// TIA Portal V17 export
// export: Created 2025-03-07T09:18:53.7752004Z, ExportSetting WithDefaults, DisplayName Totally Integrated Automation Portal, DisplayVersion V17 Update 8, DisplayName TIA Portal Openness, DisplayVersion V17 Update 8, DisplayName TIA Portal Version Control Interface, DisplayVersion V17, DisplayName SINAMICS Startdrive Advanced, DisplayVersion V17 SP2, DisplayName SINAMICS Startdrive G110M, G120, G120C, G120D, G120P, G115D, DisplayVersion V17 SP2, DisplayName SINAMICS Startdrive G130, G150, S120, S150, SINAMICS MV, S210, DisplayVersion V17 SP2, DisplayName STEP 7 Professional, DisplayVersion V17 Update 8, DisplayName SINUMERIK ONE STEP 7 Toolbox, DisplayVersion V17 Update 12, DisplayName SINUMERIK 840D sl STEP 7 Toolbox, DisplayVersion V17 Update 12, DisplayName STEP 7 Safety, DisplayVersion V17 Update 6, DisplayName WinCC Advanced, DisplayVersion V17 Update 8
FUNCTION_BLOCK "FB20200_TRUMPF_READY"   // FB20200, LAD
TITLE = FB20200 READY TRUMPF
{ S7_Optimized_Access := 'FALSE' }
VERSION : 0.1
// stored: AutoNumber false, IsIECCheckEnabled false, SetENOAutomatically false, UDAEnableTagReadback false
   VAR_INPUT
      iLIMIT_MIN_POWER : Int;   // LASER POWER MIN LIMIT
      iLIMIT_MAX_POWER : Int;   // LASER POWER MAX LIMIT
      iCOMMAND_POWER : Int;   // CNC POWER VALUE
      iCOMMAND_PROCESSING : Int;   // CNC PROCESSING VALUE
      iCOMMAND_POWER_PORTION_CORE : Int;   // CNC POWER PORTION CORE VALUE
      iSTATUS_READY_LASER_READY : Bool;   // LASER STATUS: READY
      iLASER_IS_ON : Bool;   // LASER IS ON
      iSYSTEM_ERROR_LASER_FAULT : Bool;   // LASER SYSTEM ERROR / FAULT
      iEXTERNAL_CONTROL_READY : Bool;   // LASER EXTERNAL CONTROL READY
      iPROGRAM_ACTIVE : Bool;   // LASER PROGRAM ACTIVE
      iSOURCE_ENABLED : Bool;   // -
      iCOOLING_UNIT_FLOW_PRESENT : Bool;
      iCOOLING_UNIT_OVERTEMPERATURE : Bool;
      iLASER_ENABLE_POWER_SEQ : Bool;   // -
      iLASER_DISABLE_POWER_SEQ : Bool;   // -
      iSAFETY_GATES_CLOSED_LOCKED : Bool;   // LOCAL SAFETY GATES CLOSED AND LOCKED
      iLASER_ASSIGNED : Bool;   // LASER ASSIGNED
      iMACHINE_ON : Bool;   // LOCAL MACHINE ON
      iMACHINE_ON_DELAYED : Bool;   // LOCAL MACHINE ON DELAYED
      iLASER_READY_F_CIRCUIT_BRAKER : Bool;   // LASER CIRCUIT BREAKER OK
      iLASER_WARNING_LAP_ON : Bool;   // LOCAL STATION UNIT ANY CYCLE ACTIVE
      iSTATION_UNIT_ANY_CYCLE_ACT : Bool;   // LASER ACTIVE DB START GENERAL CONDITIONS
      iLASER_ACT_START_GEN_CONDITION : Bool;
      iUNIT_NO : Byte;
   END_VAR
   VAR_OUTPUT
      oLIGHT_PATH : Byte;
      oPROGRAM_NUMBER : Byte;
      oPOWER_VALUE : DInt;
      oPROCESSING_VALUE : DInt;
      oPOWER_PORTION_CORE_VALUE : DInt;
      oLASER_RESET_FAULT_ERROR : Bool;
      oLASER_REQUEST : Bool;
      oEXTERNAL_CONTROL : Bool;
      oLASER_ON : Bool;
      oLASER_ARM : Bool;
      oSTATION_RHP_SEOC_ALARMS : Bool;
      oSTATION_WARNING : Bool;
      oREADY_TO_EMISSION : Bool;
      oALARM_CIRCUIT_BREAKER_ALARM : Bool;
      oALARM_LASER_ERROR : Bool;
      oALARM_WARNING_LASER : Bool;
      oALARM_LASER_NOT_READY : Bool;
      oALARM_LASER_NOT_SWITCHED_ON : Bool;
      oALARM_ANALOG_CONTROL_ERROR : Bool;
      oALARM_LASER_NOT_ASSIGNED : Bool;
      oALARM_OVERTEMPERATURE_ALARM : Bool;
      oALARM_LASER_EMERGENCY_STOP_ACTIVE : Bool;
      oALARM_LASER_SC_STATUS_ACTIVE : Bool;
      oALARM_ACTIVE_PANEL_ERROR : Bool;
      oALARM_LASER_MODULE_1_IN_TEST_MODE : Bool;
      oALARM_FAULT : Bool;
   END_VAR
   VAR DB_SPECIFIC
      DATA { S7_SetPoint := 'True'} : "LASER READY";
      "EXT PULSE START REQ" { S7_SetPoint := 'True'} : TON_TIME;
      "COOLING UNIT FLOW IN" : Bool;
      "COOLING OVERTEMPERATURE IN" : Bool;
      "COOLING UNIT FLOW ALARM" : Bool;
      "COOLING OVERTEMPERATURE ALARM" : Bool;
      INT_AUX : Int;
   END_VAR
   VAR_TEMP
      DB_NUMBER : DInt;
   END_VAR
   VAR_TEMP   // added for the SCL form of the ladder/FBD networks
      _w1 : Bool;
      _w2 : Bool;
      _w3 : Bool;
      _w4 : Bool;
   END_VAR
BEGIN

NETWORK
TITLE = READ INSTANCE DB NUMBER
      L     DINO;
      +     10#800000;
      T     #DB_NUMBER;

REGION Network 2: VARIABLE VALUE
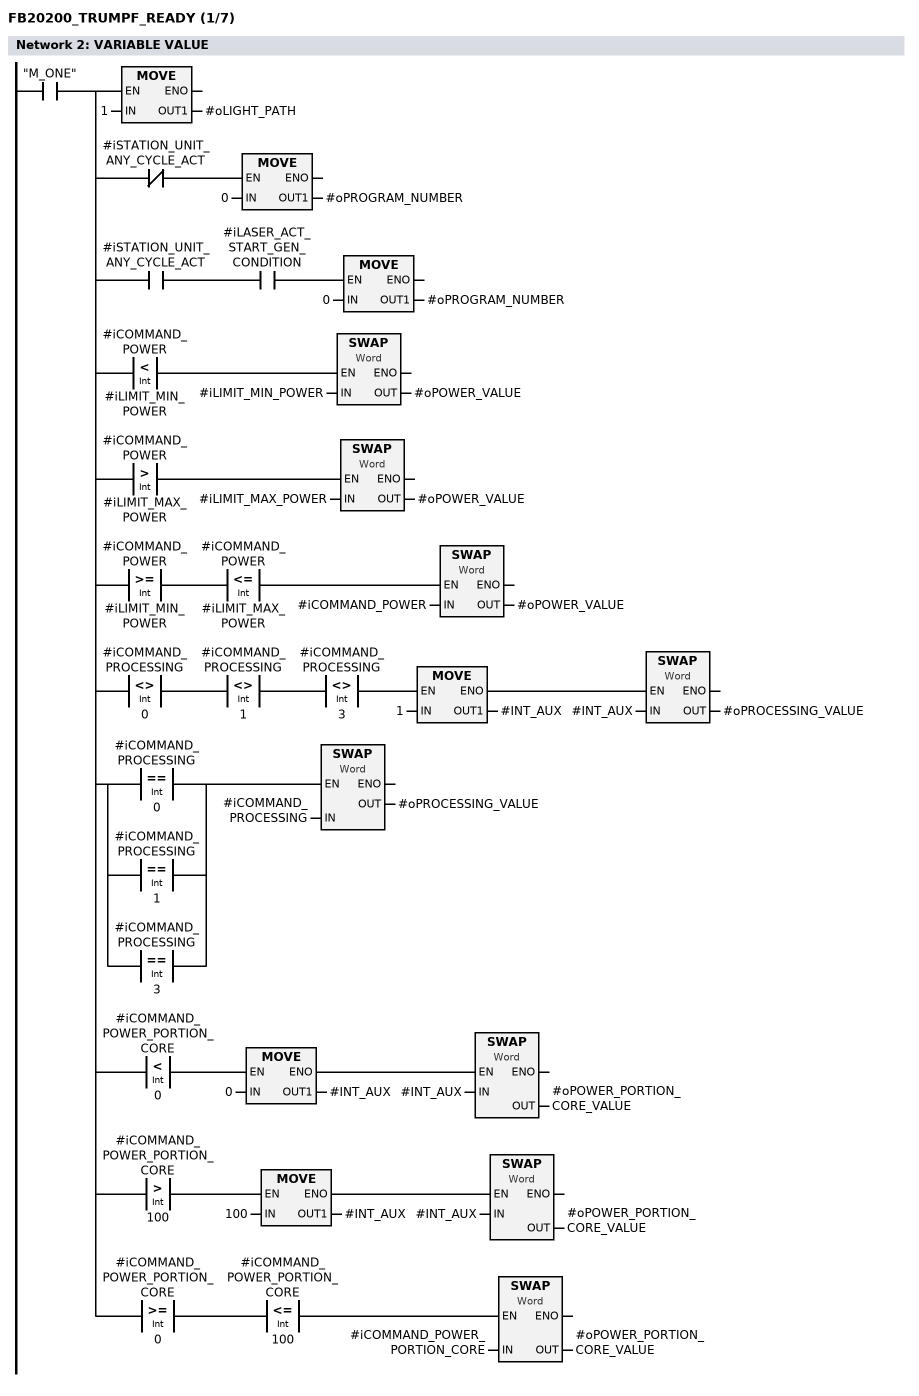
   IF "M_ONE" THEN #oLIGHT_PATH := 1; END_IF;
   IF "M_ONE" AND NOT #iSTATION_UNIT_ANY_CYCLE_ACT THEN #oPROGRAM_NUMBER := 0; END_IF;
   IF "M_ONE" AND #iSTATION_UNIT_ANY_CYCLE_ACT AND #iLASER_ACT_START_GEN_CONDITION THEN
       #oPROGRAM_NUMBER := 0;
   END_IF;
   IF "M_ONE" AND (#iCOMMAND_POWER < #iLIMIT_MIN_POWER) THEN
       #oPOWER_VALUE := SWAP(#iLIMIT_MIN_POWER);
   END_IF;
   IF "M_ONE" AND (#iCOMMAND_POWER > #iLIMIT_MAX_POWER) THEN
       #oPOWER_VALUE := SWAP(#iLIMIT_MAX_POWER);
   END_IF;
   IF "M_ONE" AND (#iCOMMAND_POWER >= #iLIMIT_MIN_POWER) AND (#iCOMMAND_POWER <= #iLIMIT_MAX_POWER) THEN
       #oPOWER_VALUE := SWAP(#iCOMMAND_POWER);
   END_IF;
   IF "M_ONE" AND (#iCOMMAND_PROCESSING <> 0) AND (#iCOMMAND_PROCESSING <> 1) AND (#iCOMMAND_PROCESSING <> 3) THEN
       #INT_AUX := 1;
       #oPROCESSING_VALUE := SWAP(#INT_AUX);
   END_IF;
   IF "M_ONE" AND ((#iCOMMAND_PROCESSING = 0) OR (#iCOMMAND_PROCESSING = 1) OR (#iCOMMAND_PROCESSING = 3)) THEN
       #oPROCESSING_VALUE := SWAP(#iCOMMAND_PROCESSING);
   END_IF;
   IF "M_ONE" AND (#iCOMMAND_POWER_PORTION_CORE < 0) THEN
       #INT_AUX := 0;
       #oPOWER_PORTION_CORE_VALUE := SWAP(#INT_AUX);
   END_IF;
   IF "M_ONE" AND (#iCOMMAND_POWER_PORTION_CORE > 100) THEN
       #INT_AUX := 100;
       #oPOWER_PORTION_CORE_VALUE := SWAP(#INT_AUX);
   END_IF;
   IF "M_ONE" AND (#iCOMMAND_POWER_PORTION_CORE >= 0) AND (#iCOMMAND_POWER_PORTION_CORE <= 100) THEN
       #oPOWER_PORTION_CORE_VALUE := SWAP(#iCOMMAND_POWER_PORTION_CORE);
   END_IF;
END_REGION

REGION Network 3: INPUT
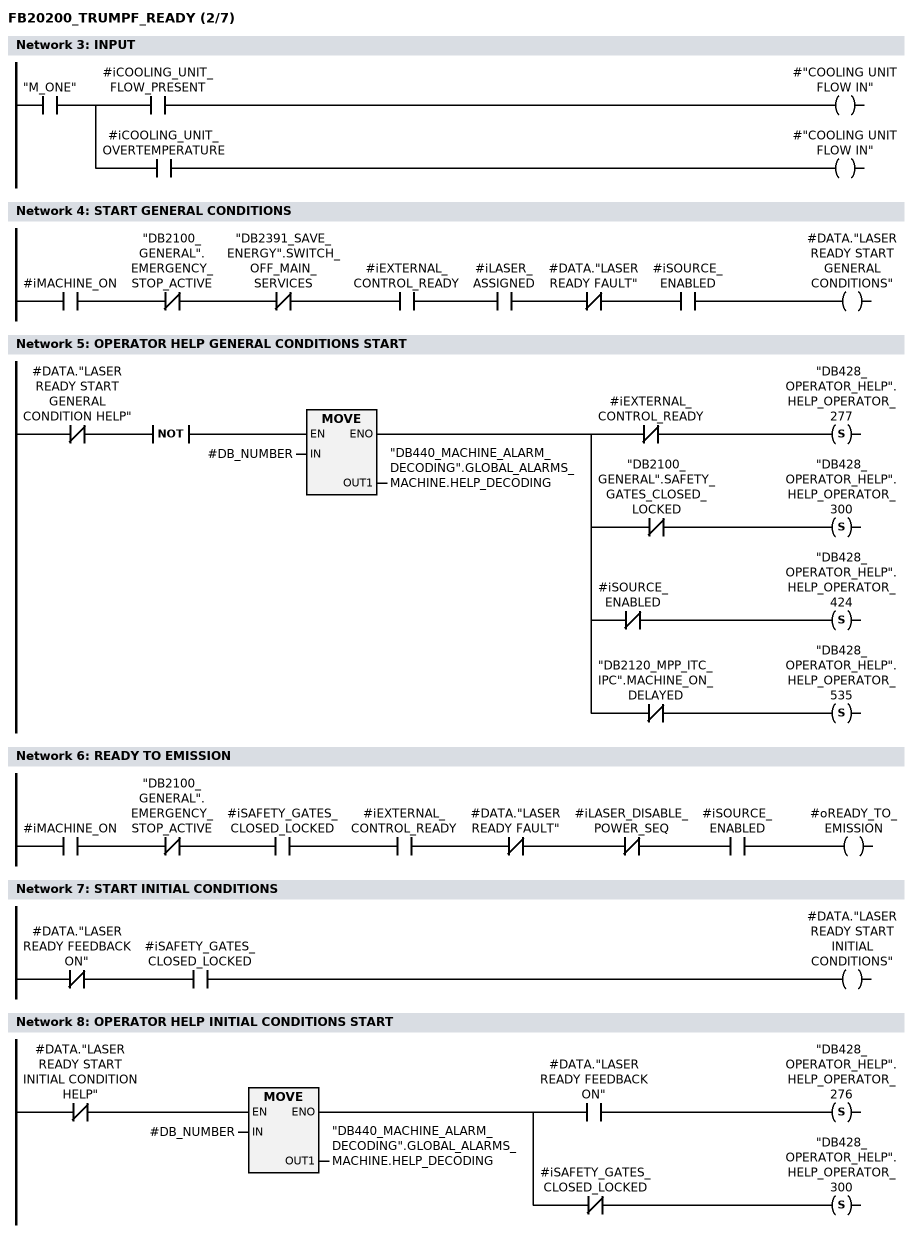
   RUNG wire#powerrail
      Contact( "M_ONE" )
      wire#w1
      Contact( #iCOOLING_UNIT_FLOW_PRESENT )
      Coil( #"COOLING UNIT FLOW IN" )
   END_RUNG
   RUNG wire#w1
      Contact( #iCOOLING_UNIT_OVERTEMPERATURE )
      Coil( #"COOLING UNIT FLOW IN" )
   END_RUNG
   // the same network as SCL:
   #"COOLING UNIT FLOW IN" := "M_ONE" AND #iCOOLING_UNIT_FLOW_PRESENT;
   #"COOLING UNIT FLOW IN" := "M_ONE" AND #iCOOLING_UNIT_OVERTEMPERATURE;
END_REGION

REGION Network 4: START GENERAL CONDITIONS
   RUNG wire#powerrail
      Contact( #iMACHINE_ON )
      I_Contact( "DB2100_GENERAL".EMERGENCY_STOP_ACTIVE )
      I_Contact( "DB2391_SAVE_ENERGY".SWITCH_OFF_MAIN_SERVICES )
      Contact( #iEXTERNAL_CONTROL_READY )
      Contact( #iLASER_ASSIGNED )
      I_Contact( #DATA."LASER READY FAULT" )
      Contact( #iSOURCE_ENABLED )
      Coil( #DATA."LASER READY START GENERAL CONDITIONS" )
   END_RUNG
   // the same network as SCL:
   #DATA."LASER READY START GENERAL CONDITIONS" := #iMACHINE_ON AND NOT "DB2100_GENERAL".EMERGENCY_STOP_ACTIVE AND NOT "DB2391_SAVE_ENERGY".SWITCH_OFF_MAIN_SERVICES AND #iEXTERNAL_CONTROL_READY AND #iLASER_ASSIGNED AND NOT #DATA."LASER READY FAULT" AND #iSOURCE_ENABLED;
END_REGION

REGION Network 5: OPERATOR HELP GENERAL CONDITIONS START
   RUNG wire#powerrail
      I_Contact( #DATA."LASER READY START GENERAL CONDITION HELP" )
      Not()
      Move(in := #DB_NUMBER, out1 => "DB440_MACHINE_ALARM_DECODING".GLOBAL_ALARMS_MACHINE.HELP_DECODING)
      wire#w1
      I_Contact( #iEXTERNAL_CONTROL_READY )
      S_Coil( "DB428_OPERATOR_HELP".HELP_OPERATOR_277 )
   END_RUNG
   RUNG wire#w1
      I_Contact( "DB2100_GENERAL".SAFETY_GATES_CLOSED_LOCKED )
      S_Coil( "DB428_OPERATOR_HELP".HELP_OPERATOR_300 )
   END_RUNG
   RUNG wire#w1
      I_Contact( #iSOURCE_ENABLED )
      S_Coil( "DB428_OPERATOR_HELP".HELP_OPERATOR_424 )
   END_RUNG
   RUNG wire#w1
      I_Contact( "DB2120_MPP_ITC_IPC".MACHINE_ON_DELAYED )
      S_Coil( "DB428_OPERATOR_HELP".HELP_OPERATOR_535 )
   END_RUNG
   // the same network as SCL:
   #_w1 := NOT (NOT #DATA."LASER READY START GENERAL CONDITION HELP");
   IF #_w1 THEN "DB440_MACHINE_ALARM_DECODING".GLOBAL_ALARMS_MACHINE.HELP_DECODING := #DB_NUMBER; END_IF;
   IF #_w1 AND NOT #iEXTERNAL_CONTROL_READY THEN "DB428_OPERATOR_HELP".HELP_OPERATOR_277 := TRUE; END_IF;
   IF #_w1 AND NOT "DB2100_GENERAL".SAFETY_GATES_CLOSED_LOCKED THEN
       "DB428_OPERATOR_HELP".HELP_OPERATOR_300 := TRUE;
   END_IF;
   IF #_w1 AND NOT #iSOURCE_ENABLED THEN "DB428_OPERATOR_HELP".HELP_OPERATOR_424 := TRUE; END_IF;
   IF #_w1 AND NOT "DB2120_MPP_ITC_IPC".MACHINE_ON_DELAYED THEN
       "DB428_OPERATOR_HELP".HELP_OPERATOR_535 := TRUE;
   END_IF;
END_REGION

REGION Network 6: READY TO EMISSION
   RUNG wire#powerrail
      Contact( #iMACHINE_ON )
      I_Contact( "DB2100_GENERAL".EMERGENCY_STOP_ACTIVE )
      Contact( #iSAFETY_GATES_CLOSED_LOCKED )
      Contact( #iEXTERNAL_CONTROL_READY )
      I_Contact( #DATA."LASER READY FAULT" )
      I_Contact( #iLASER_DISABLE_POWER_SEQ )
      Contact( #iSOURCE_ENABLED )
      Coil( #oREADY_TO_EMISSION )
   END_RUNG
   // the same network as SCL:
   #oREADY_TO_EMISSION := #iMACHINE_ON AND NOT "DB2100_GENERAL".EMERGENCY_STOP_ACTIVE AND #iSAFETY_GATES_CLOSED_LOCKED AND #iEXTERNAL_CONTROL_READY AND NOT #DATA."LASER READY FAULT" AND NOT #iLASER_DISABLE_POWER_SEQ AND #iSOURCE_ENABLED;
END_REGION

REGION Network 7: START INITIAL CONDITIONS
   RUNG wire#powerrail
      I_Contact( #DATA."LASER READY FEEDBACK ON" )
      Contact( #iSAFETY_GATES_CLOSED_LOCKED )
      Coil( #DATA."LASER READY START INITIAL CONDITIONS" )
   END_RUNG
   // the same network as SCL:
   #DATA."LASER READY START INITIAL CONDITIONS" := NOT #DATA."LASER READY FEEDBACK ON" AND #iSAFETY_GATES_CLOSED_LOCKED;
END_REGION

REGION Network 8: OPERATOR HELP INITIAL CONDITIONS START
   RUNG wire#powerrail
      I_Contact( #DATA."LASER READY START INITIAL CONDITION HELP" )
      Move(in := #DB_NUMBER, out1 => "DB440_MACHINE_ALARM_DECODING".GLOBAL_ALARMS_MACHINE.HELP_DECODING)
      wire#w1
      Contact( #DATA."LASER READY FEEDBACK ON" )
      S_Coil( "DB428_OPERATOR_HELP".HELP_OPERATOR_276 )
   END_RUNG
   RUNG wire#w1
      I_Contact( #iSAFETY_GATES_CLOSED_LOCKED )
      S_Coil( "DB428_OPERATOR_HELP".HELP_OPERATOR_300 )
   END_RUNG
   // the same network as SCL:
   #_w1 := NOT #DATA."LASER READY START INITIAL CONDITION HELP";
   IF #_w1 THEN "DB440_MACHINE_ALARM_DECODING".GLOBAL_ALARMS_MACHINE.HELP_DECODING := #DB_NUMBER; END_IF;
   IF #_w1 AND #DATA."LASER READY FEEDBACK ON" THEN "DB428_OPERATOR_HELP".HELP_OPERATOR_276 := TRUE; END_IF;
   IF #_w1 AND NOT #iSAFETY_GATES_CLOSED_LOCKED THEN "DB428_OPERATOR_HELP".HELP_OPERATOR_300 := TRUE; END_IF;
END_REGION

REGION Network 9: AUTO START REQUEST
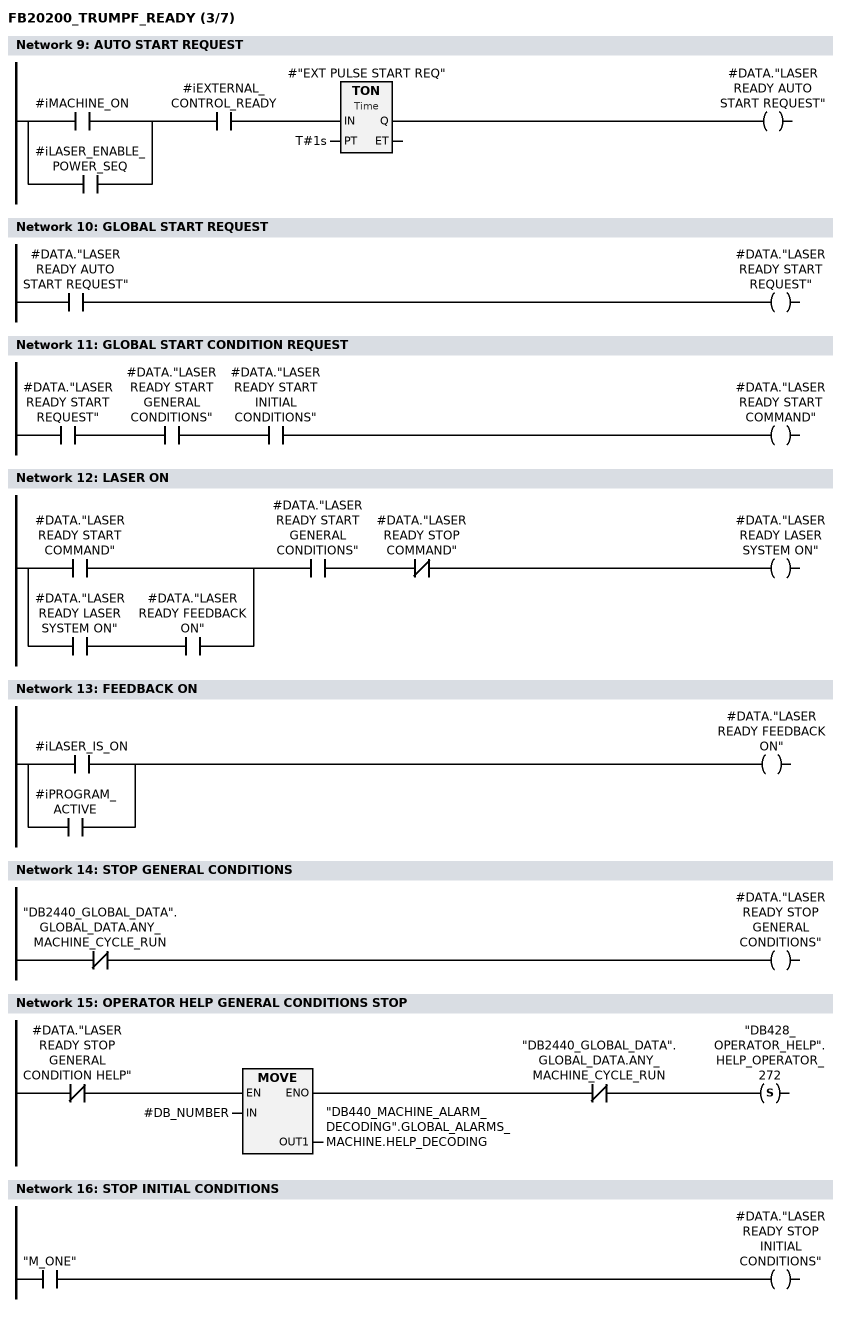
   RUNG wire#powerrail
      Contact( #iMACHINE_ON )
      wire#w1
      Contact( #iEXTERNAL_CONTROL_READY )
      { S7_Templates := "time_type := Time" } #"EXT PULSE START REQ".TON(pt := T#1s, et =>)
      Coil( #DATA."LASER READY AUTO START REQUEST" )
   END_RUNG
   RUNG wire#powerrail
      Contact( #iLASER_ENABLE_POWER_SEQ )
   END_RUNG wire#w1
   // the same network as SCL:
   #"EXT PULSE START REQ"(IN := (#iMACHINE_ON OR #iLASER_ENABLE_POWER_SEQ) AND #iEXTERNAL_CONTROL_READY,   // TON
                          PT := T#1s);
   #DATA."LASER READY AUTO START REQUEST" := #"EXT PULSE START REQ".Q;
END_REGION

REGION Network 10: GLOBAL START REQUEST
   RUNG wire#powerrail
      Contact( #DATA."LASER READY AUTO START REQUEST" )
      Coil( #DATA."LASER READY START REQUEST" )
   END_RUNG
   // the same network as SCL:
   #DATA."LASER READY START REQUEST" := #DATA."LASER READY AUTO START REQUEST";
END_REGION

REGION Network 11: GLOBAL START CONDITION REQUEST
   RUNG wire#powerrail
      Contact( #DATA."LASER READY START REQUEST" )
      Contact( #DATA."LASER READY START GENERAL CONDITIONS" )
      Contact( #DATA."LASER READY START INITIAL CONDITIONS" )
      Coil( #DATA."LASER READY START COMMAND" )
   END_RUNG
   // the same network as SCL:
   #DATA."LASER READY START COMMAND" := #DATA."LASER READY START REQUEST" AND #DATA."LASER READY START GENERAL CONDITIONS" AND #DATA."LASER READY START INITIAL CONDITIONS";
END_REGION

REGION Network 12: LASER ON
   RUNG wire#powerrail
      Contact( #DATA."LASER READY START COMMAND" )
      wire#w1
      Contact( #DATA."LASER READY START GENERAL CONDITIONS" )
      I_Contact( #DATA."LASER READY STOP COMMAND" )
      Coil( #DATA."LASER READY LASER SYSTEM ON" )
   END_RUNG
   RUNG wire#powerrail
      Contact( #DATA."LASER READY LASER SYSTEM ON" )
      Contact( #DATA."LASER READY FEEDBACK ON" )
   END_RUNG wire#w1
   // the same network as SCL:
   #DATA."LASER READY LASER SYSTEM ON" := (#DATA."LASER READY START COMMAND" OR (#DATA."LASER READY LASER SYSTEM ON" AND #DATA."LASER READY FEEDBACK ON")) AND #DATA."LASER READY START GENERAL CONDITIONS" AND NOT #DATA."LASER READY STOP COMMAND";
END_REGION

REGION Network 13: FEEDBACK ON
   RUNG wire#powerrail
      Contact( #iLASER_IS_ON )
      wire#w1
      Coil( #DATA."LASER READY FEEDBACK ON" )
   END_RUNG
   RUNG wire#powerrail
      Contact( #iPROGRAM_ACTIVE )
   END_RUNG wire#w1
   // the same network as SCL:
   #DATA."LASER READY FEEDBACK ON" := #iLASER_IS_ON OR #iPROGRAM_ACTIVE;
END_REGION

REGION Network 14: STOP GENERAL CONDITIONS
   RUNG wire#powerrail
      I_Contact( "DB2440_GLOBAL_DATA".GLOBAL_DATA.ANY_MACHINE_CYCLE_RUN )
      Coil( #DATA."LASER READY STOP GENERAL CONDITIONS" )
   END_RUNG
   // the same network as SCL:
   #DATA."LASER READY STOP GENERAL CONDITIONS" := NOT "DB2440_GLOBAL_DATA".GLOBAL_DATA.ANY_MACHINE_CYCLE_RUN;
END_REGION

REGION Network 15: OPERATOR HELP GENERAL CONDITIONS STOP
   RUNG wire#powerrail
      I_Contact( #DATA."LASER READY STOP GENERAL CONDITION HELP" )
      Move(in := #DB_NUMBER, out1 => "DB440_MACHINE_ALARM_DECODING".GLOBAL_ALARMS_MACHINE.HELP_DECODING)
      I_Contact( "DB2440_GLOBAL_DATA".GLOBAL_DATA.ANY_MACHINE_CYCLE_RUN )
      S_Coil( "DB428_OPERATOR_HELP".HELP_OPERATOR_272 )
   END_RUNG
   // the same network as SCL:
   #_w1 := NOT #DATA."LASER READY STOP GENERAL CONDITION HELP";
   IF #_w1 THEN "DB440_MACHINE_ALARM_DECODING".GLOBAL_ALARMS_MACHINE.HELP_DECODING := #DB_NUMBER; END_IF;
   IF #_w1 AND NOT "DB2440_GLOBAL_DATA".GLOBAL_DATA.ANY_MACHINE_CYCLE_RUN THEN
       "DB428_OPERATOR_HELP".HELP_OPERATOR_272 := TRUE;
   END_IF;
END_REGION

REGION Network 16: STOP INITIAL CONDITIONS
   RUNG wire#powerrail
      Contact( "M_ONE" )
      Coil( #DATA."LASER READY STOP INITIAL CONDITIONS" )
   END_RUNG
   // the same network as SCL:
   #DATA."LASER READY STOP INITIAL CONDITIONS" := "M_ONE";
END_REGION

REGION Network 17: OPERATOR HELP INITIAL CONDITIONS STOP
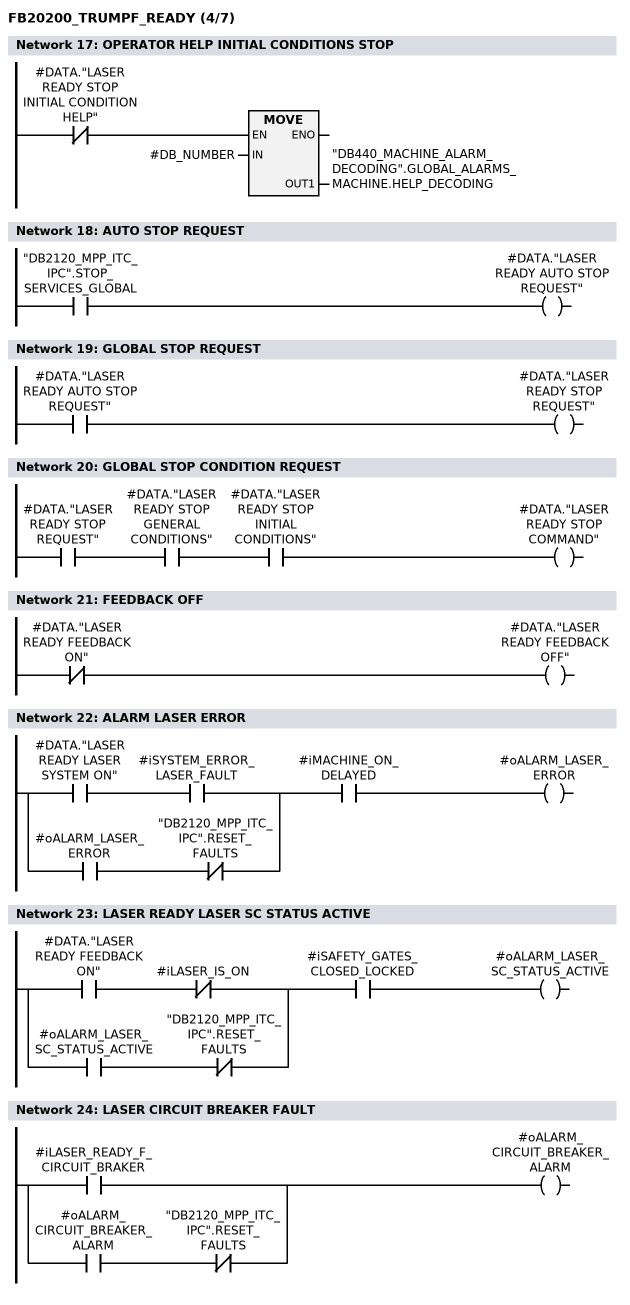
   RUNG wire#powerrail
      I_Contact( #DATA."LASER READY STOP INITIAL CONDITION HELP" )
      Move(in := #DB_NUMBER, out1 => "DB440_MACHINE_ALARM_DECODING".GLOBAL_ALARMS_MACHINE.HELP_DECODING)
   END_RUNG
   // the same network as SCL:
   IF NOT #DATA."LASER READY STOP INITIAL CONDITION HELP" THEN
       "DB440_MACHINE_ALARM_DECODING".GLOBAL_ALARMS_MACHINE.HELP_DECODING := #DB_NUMBER;
   END_IF;
END_REGION

REGION Network 18: AUTO STOP REQUEST
   RUNG wire#powerrail
      Contact( "DB2120_MPP_ITC_IPC".STOP_SERVICES_GLOBAL )
      Coil( #DATA."LASER READY AUTO STOP REQUEST" )
   END_RUNG
   // the same network as SCL:
   #DATA."LASER READY AUTO STOP REQUEST" := "DB2120_MPP_ITC_IPC".STOP_SERVICES_GLOBAL;
END_REGION

REGION Network 19: GLOBAL STOP REQUEST
   RUNG wire#powerrail
      Contact( #DATA."LASER READY AUTO STOP REQUEST" )
      Coil( #DATA."LASER READY STOP REQUEST" )
   END_RUNG
   // the same network as SCL:
   #DATA."LASER READY STOP REQUEST" := #DATA."LASER READY AUTO STOP REQUEST";
END_REGION

REGION Network 20: GLOBAL STOP CONDITION REQUEST
   RUNG wire#powerrail
      Contact( #DATA."LASER READY STOP REQUEST" )
      Contact( #DATA."LASER READY STOP GENERAL CONDITIONS" )
      Contact( #DATA."LASER READY STOP INITIAL CONDITIONS" )
      Coil( #DATA."LASER READY STOP COMMAND" )
   END_RUNG
   // the same network as SCL:
   #DATA."LASER READY STOP COMMAND" := #DATA."LASER READY STOP REQUEST" AND #DATA."LASER READY STOP GENERAL CONDITIONS" AND #DATA."LASER READY STOP INITIAL CONDITIONS";
END_REGION

REGION Network 21: FEEDBACK OFF
   RUNG wire#powerrail
      I_Contact( #DATA."LASER READY FEEDBACK ON" )
      Coil( #DATA."LASER READY FEEDBACK OFF" )
   END_RUNG
   // the same network as SCL:
   #DATA."LASER READY FEEDBACK OFF" := NOT #DATA."LASER READY FEEDBACK ON";
END_REGION

REGION Network 22: ALARM LASER ERROR
   RUNG wire#powerrail
      Contact( #DATA."LASER READY LASER SYSTEM ON" )
      Contact( #iSYSTEM_ERROR_LASER_FAULT )
      wire#w1
      Contact( #iMACHINE_ON_DELAYED )
      Coil( #oALARM_LASER_ERROR )
   END_RUNG
   RUNG wire#powerrail
      Contact( #oALARM_LASER_ERROR )
      I_Contact( "DB2120_MPP_ITC_IPC".RESET_FAULTS )
   END_RUNG wire#w1
   // the same network as SCL:
   #oALARM_LASER_ERROR := ((#DATA."LASER READY LASER SYSTEM ON" AND #iSYSTEM_ERROR_LASER_FAULT) OR (#oALARM_LASER_ERROR AND NOT "DB2120_MPP_ITC_IPC".RESET_FAULTS)) AND #iMACHINE_ON_DELAYED;
END_REGION

REGION Network 23: LASER READY LASER SC STATUS ACTIVE
   RUNG wire#powerrail
      Contact( #DATA."LASER READY FEEDBACK ON" )
      I_Contact( #iLASER_IS_ON )
      wire#w1
      Contact( #iSAFETY_GATES_CLOSED_LOCKED )
      Coil( #oALARM_LASER_SC_STATUS_ACTIVE )
   END_RUNG
   RUNG wire#powerrail
      Contact( #oALARM_LASER_SC_STATUS_ACTIVE )
      I_Contact( "DB2120_MPP_ITC_IPC".RESET_FAULTS )
   END_RUNG wire#w1
   // the same network as SCL:
   #oALARM_LASER_SC_STATUS_ACTIVE := ((#DATA."LASER READY FEEDBACK ON" AND NOT #iLASER_IS_ON) OR (#oALARM_LASER_SC_STATUS_ACTIVE AND NOT "DB2120_MPP_ITC_IPC".RESET_FAULTS)) AND #iSAFETY_GATES_CLOSED_LOCKED;
END_REGION

REGION Network 24: LASER CIRCUIT BREAKER FAULT
   RUNG wire#powerrail
      Contact( #iLASER_READY_F_CIRCUIT_BRAKER )
      wire#w1
      Coil( #oALARM_CIRCUIT_BREAKER_ALARM )
   END_RUNG
   RUNG wire#powerrail
      Contact( #oALARM_CIRCUIT_BREAKER_ALARM )
      I_Contact( "DB2120_MPP_ITC_IPC".RESET_FAULTS )
   END_RUNG wire#w1
   // the same network as SCL:
   #oALARM_CIRCUIT_BREAKER_ALARM := #iLASER_READY_F_CIRCUIT_BRAKER OR (#oALARM_CIRCUIT_BREAKER_ALARM AND NOT "DB2120_MPP_ITC_IPC".RESET_FAULTS);
END_REGION

REGION Network 25: LASER NOT READY
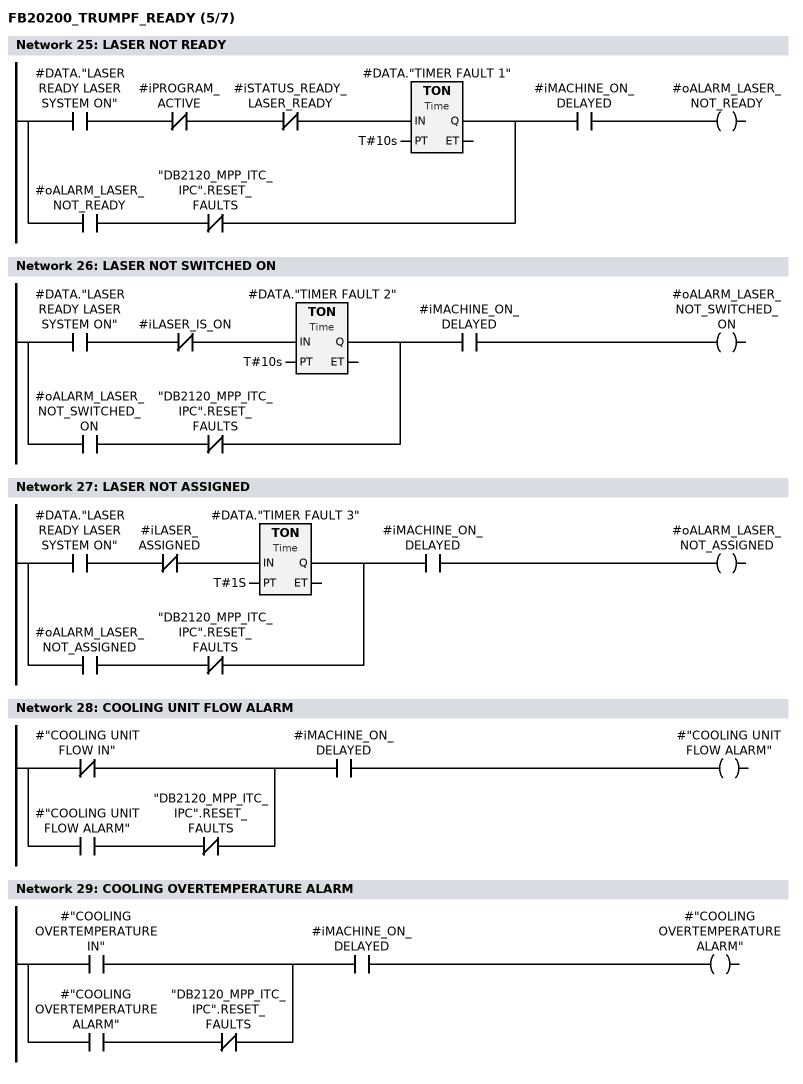
   RUNG wire#powerrail
      Contact( #DATA."LASER READY LASER SYSTEM ON" )
      I_Contact( #iPROGRAM_ACTIVE )
      I_Contact( #iSTATUS_READY_LASER_READY )
      { S7_Templates := "time_type := Time" } #DATA."TIMER FAULT 1".TON(pt := T#10s, et =>)
      wire#w1
      Contact( #iMACHINE_ON_DELAYED )
      Coil( #oALARM_LASER_NOT_READY )
   END_RUNG
   RUNG wire#powerrail
      Contact( #oALARM_LASER_NOT_READY )
      I_Contact( "DB2120_MPP_ITC_IPC".RESET_FAULTS )
   END_RUNG wire#w1
   // the same network as SCL:
   #DATA."TIMER FAULT 1".TON(IN := #DATA."LASER READY LASER SYSTEM ON" AND NOT #iPROGRAM_ACTIVE AND NOT #iSTATUS_READY_LASER_READY,
                           PT := T#10s);
   #oALARM_LASER_NOT_READY := (#DATA."TIMER FAULT 1".Q OR (#oALARM_LASER_NOT_READY AND NOT "DB2120_MPP_ITC_IPC".RESET_FAULTS)) AND #iMACHINE_ON_DELAYED;
END_REGION

REGION Network 26: LASER NOT SWITCHED ON
   RUNG wire#powerrail
      Contact( #DATA."LASER READY LASER SYSTEM ON" )
      I_Contact( #iLASER_IS_ON )
      { S7_Templates := "time_type := Time" } #DATA."TIMER FAULT 2".TON(pt := T#10s, et =>)
      wire#w1
      Contact( #iMACHINE_ON_DELAYED )
      Coil( #oALARM_LASER_NOT_SWITCHED_ON )
   END_RUNG
   RUNG wire#powerrail
      Contact( #oALARM_LASER_NOT_SWITCHED_ON )
      I_Contact( "DB2120_MPP_ITC_IPC".RESET_FAULTS )
   END_RUNG wire#w1
   // the same network as SCL:
   #DATA."TIMER FAULT 2".TON(IN := #DATA."LASER READY LASER SYSTEM ON" AND NOT #iLASER_IS_ON, PT := T#10s);
   #oALARM_LASER_NOT_SWITCHED_ON := (#DATA."TIMER FAULT 2".Q OR (#oALARM_LASER_NOT_SWITCHED_ON AND NOT "DB2120_MPP_ITC_IPC".RESET_FAULTS)) AND #iMACHINE_ON_DELAYED;
END_REGION

REGION Network 27: LASER NOT ASSIGNED
   RUNG wire#powerrail
      Contact( #DATA."LASER READY LASER SYSTEM ON" )
      I_Contact( #iLASER_ASSIGNED )
      { S7_Templates := "time_type := Time" } #DATA."TIMER FAULT 3".TON(pt := T#1S, et =>)
      wire#w1
      Contact( #iMACHINE_ON_DELAYED )
      Coil( #oALARM_LASER_NOT_ASSIGNED )
   END_RUNG
   RUNG wire#powerrail
      Contact( #oALARM_LASER_NOT_ASSIGNED )
      I_Contact( "DB2120_MPP_ITC_IPC".RESET_FAULTS )
   END_RUNG wire#w1
   // the same network as SCL:
   #DATA."TIMER FAULT 3".TON(IN := #DATA."LASER READY LASER SYSTEM ON" AND NOT #iLASER_ASSIGNED, PT := T#1S);
   #oALARM_LASER_NOT_ASSIGNED := (#DATA."TIMER FAULT 3".Q OR (#oALARM_LASER_NOT_ASSIGNED AND NOT "DB2120_MPP_ITC_IPC".RESET_FAULTS)) AND #iMACHINE_ON_DELAYED;
END_REGION

REGION Network 28: COOLING UNIT FLOW ALARM
   RUNG wire#powerrail
      I_Contact( #"COOLING UNIT FLOW IN" )
      wire#w1
      Contact( #iMACHINE_ON_DELAYED )
      Coil( #"COOLING UNIT FLOW ALARM" )
   END_RUNG
   RUNG wire#powerrail
      Contact( #"COOLING UNIT FLOW ALARM" )
      I_Contact( "DB2120_MPP_ITC_IPC".RESET_FAULTS )
   END_RUNG wire#w1
   // the same network as SCL:
   #"COOLING UNIT FLOW ALARM" := (NOT #"COOLING UNIT FLOW IN" OR (#"COOLING UNIT FLOW ALARM" AND NOT "DB2120_MPP_ITC_IPC".RESET_FAULTS)) AND #iMACHINE_ON_DELAYED;
END_REGION

REGION Network 29: COOLING OVERTEMPERATURE ALARM
   RUNG wire#powerrail
      Contact( #"COOLING OVERTEMPERATURE IN" )
      wire#w1
      Contact( #iMACHINE_ON_DELAYED )
      Coil( #"COOLING OVERTEMPERATURE ALARM" )
   END_RUNG
   RUNG wire#powerrail
      Contact( #"COOLING OVERTEMPERATURE ALARM" )
      I_Contact( "DB2120_MPP_ITC_IPC".RESET_FAULTS )
   END_RUNG wire#w1
   // the same network as SCL:
   #"COOLING OVERTEMPERATURE ALARM" := (#"COOLING OVERTEMPERATURE IN" OR (#"COOLING OVERTEMPERATURE ALARM" AND NOT "DB2120_MPP_ITC_IPC".RESET_FAULTS)) AND #iMACHINE_ON_DELAYED;
END_REGION

REGION Network 30: RETURN HOME POSITION AND STOP END OF CYCLE ALARMS
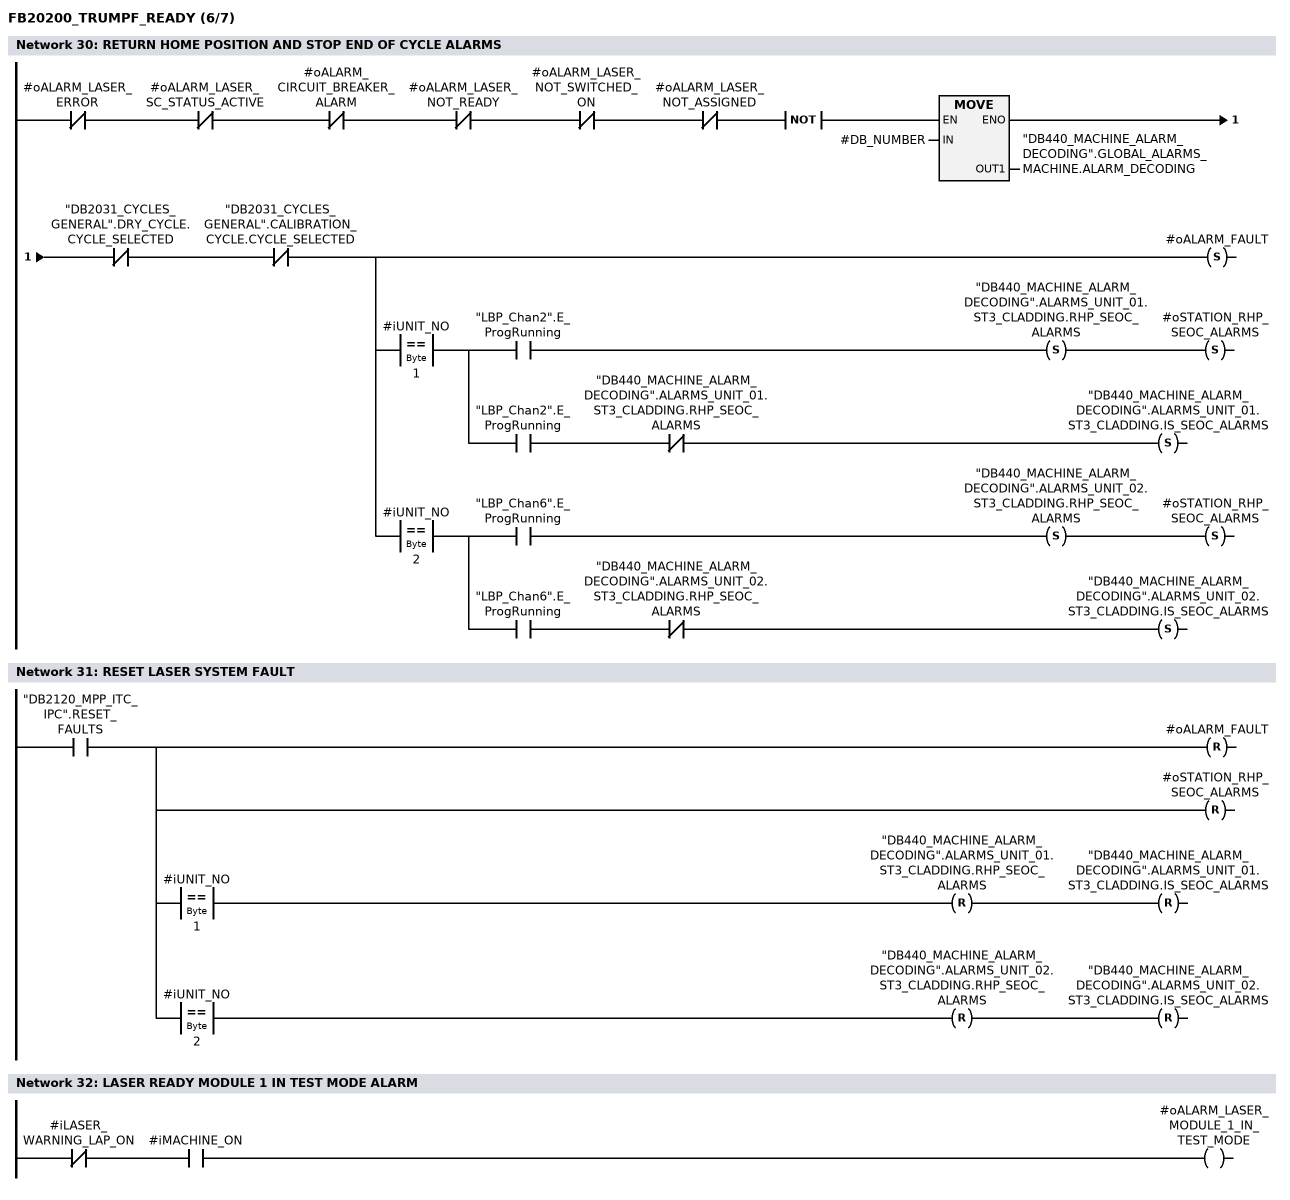
   RUNG wire#powerrail
      I_Contact( #oALARM_LASER_ERROR )
      I_Contact( #oALARM_LASER_SC_STATUS_ACTIVE )
      I_Contact( #oALARM_CIRCUIT_BREAKER_ALARM )
      I_Contact( #oALARM_LASER_NOT_READY )
      I_Contact( #oALARM_LASER_NOT_SWITCHED_ON )
      I_Contact( #oALARM_LASER_NOT_ASSIGNED )
      Not()
      Move(in := #DB_NUMBER, out1 => "DB440_MACHINE_ALARM_DECODING".GLOBAL_ALARMS_MACHINE.ALARM_DECODING)
      I_Contact( "DB2031_CYCLES_GENERAL".DRY_CYCLE.CYCLE_SELECTED )
      I_Contact( "DB2031_CYCLES_GENERAL".CALIBRATION_CYCLE.CYCLE_SELECTED )
      wire#w1
      S_Coil( #oALARM_FAULT )
   END_RUNG
   RUNG wire#w1
      { S7_Templates := "SrcType := Byte" } EQ_Contact(in1 := #iUNIT_NO, in2 := 1)
      wire#w2
      Contact( "LBP_Chan2".E_ProgRunning )
      S_Coil( "DB440_MACHINE_ALARM_DECODING".ALARMS_UNIT_01.ST3_CLADDING.RHP_SEOC_ALARMS )
      S_Coil( #oSTATION_RHP_SEOC_ALARMS )
   END_RUNG
   RUNG wire#w2
      Contact( "LBP_Chan2".E_ProgRunning )
      I_Contact( "DB440_MACHINE_ALARM_DECODING".ALARMS_UNIT_01.ST3_CLADDING.RHP_SEOC_ALARMS )
      S_Coil( "DB440_MACHINE_ALARM_DECODING".ALARMS_UNIT_01.ST3_CLADDING.IS_SEOC_ALARMS )
   END_RUNG
   RUNG wire#w1
      { S7_Templates := "SrcType := Byte" } EQ_Contact(in1 := #iUNIT_NO, in2 := 2)
      wire#w3
      Contact( "LBP_Chan6".E_ProgRunning )
      S_Coil( "DB440_MACHINE_ALARM_DECODING".ALARMS_UNIT_02.ST3_CLADDING.RHP_SEOC_ALARMS )
      S_Coil( #oSTATION_RHP_SEOC_ALARMS )
   END_RUNG
   RUNG wire#w3
      Contact( "LBP_Chan6".E_ProgRunning )
      I_Contact( "DB440_MACHINE_ALARM_DECODING".ALARMS_UNIT_02.ST3_CLADDING.RHP_SEOC_ALARMS )
      S_Coil( "DB440_MACHINE_ALARM_DECODING".ALARMS_UNIT_02.ST3_CLADDING.IS_SEOC_ALARMS )
   END_RUNG
   // the same network as SCL:
   #_w1 := NOT (NOT #oALARM_LASER_ERROR AND NOT #oALARM_LASER_SC_STATUS_ACTIVE AND NOT #oALARM_CIRCUIT_BREAKER_ALARM AND NOT #oALARM_LASER_NOT_READY AND NOT #oALARM_LASER_NOT_SWITCHED_ON AND NOT #oALARM_LASER_NOT_ASSIGNED);
   IF #_w1 THEN "DB440_MACHINE_ALARM_DECODING".GLOBAL_ALARMS_MACHINE.ALARM_DECODING := #DB_NUMBER; END_IF;
   #_w2 := #_w1 AND NOT "DB2031_CYCLES_GENERAL".DRY_CYCLE.CYCLE_SELECTED AND NOT "DB2031_CYCLES_GENERAL".CALIBRATION_CYCLE.CYCLE_SELECTED;
   IF #_w2 THEN #oALARM_FAULT := TRUE; END_IF;
   #_w3 := #_w2 AND (#iUNIT_NO = 1);
   IF #_w3 AND "LBP_Chan2".E_ProgRunning THEN
       "DB440_MACHINE_ALARM_DECODING".ALARMS_UNIT_01.ST3_CLADDING.RHP_SEOC_ALARMS := TRUE;
       #oSTATION_RHP_SEOC_ALARMS := TRUE;
   END_IF;
   IF #_w3 AND "LBP_Chan2".E_ProgRunning AND NOT "DB440_MACHINE_ALARM_DECODING".ALARMS_UNIT_01.ST3_CLADDING.RHP_SEOC_ALARMS THEN
       "DB440_MACHINE_ALARM_DECODING".ALARMS_UNIT_01.ST3_CLADDING.IS_SEOC_ALARMS := TRUE;
   END_IF;
   #_w4 := #_w2 AND (#iUNIT_NO = 2);
   IF #_w4 AND "LBP_Chan6".E_ProgRunning THEN
       "DB440_MACHINE_ALARM_DECODING".ALARMS_UNIT_02.ST3_CLADDING.RHP_SEOC_ALARMS := TRUE;
       #oSTATION_RHP_SEOC_ALARMS := TRUE;
   END_IF;
   IF #_w4 AND "LBP_Chan6".E_ProgRunning AND NOT "DB440_MACHINE_ALARM_DECODING".ALARMS_UNIT_02.ST3_CLADDING.RHP_SEOC_ALARMS THEN
       "DB440_MACHINE_ALARM_DECODING".ALARMS_UNIT_02.ST3_CLADDING.IS_SEOC_ALARMS := TRUE;
   END_IF;
END_REGION

REGION Network 31: RESET LASER SYSTEM FAULT
   RUNG wire#powerrail
      Contact( "DB2120_MPP_ITC_IPC".RESET_FAULTS )
      wire#w1
      R_Coil( #oALARM_FAULT )
   END_RUNG
   RUNG wire#w1
      R_Coil( #oSTATION_RHP_SEOC_ALARMS )
   END_RUNG
   RUNG wire#w1
      { S7_Templates := "SrcType := Byte" } EQ_Contact(in1 := #iUNIT_NO, in2 := 1)
      R_Coil( "DB440_MACHINE_ALARM_DECODING".ALARMS_UNIT_01.ST3_CLADDING.RHP_SEOC_ALARMS )
      R_Coil( "DB440_MACHINE_ALARM_DECODING".ALARMS_UNIT_01.ST3_CLADDING.IS_SEOC_ALARMS )
   END_RUNG
   RUNG wire#w1
      { S7_Templates := "SrcType := Byte" } EQ_Contact(in1 := #iUNIT_NO, in2 := 2)
      R_Coil( "DB440_MACHINE_ALARM_DECODING".ALARMS_UNIT_02.ST3_CLADDING.RHP_SEOC_ALARMS )
      R_Coil( "DB440_MACHINE_ALARM_DECODING".ALARMS_UNIT_02.ST3_CLADDING.IS_SEOC_ALARMS )
   END_RUNG
   // the same network as SCL:
   IF "DB2120_MPP_ITC_IPC".RESET_FAULTS THEN
       #oALARM_FAULT := FALSE;
       #oSTATION_RHP_SEOC_ALARMS := FALSE;
   END_IF;
   IF "DB2120_MPP_ITC_IPC".RESET_FAULTS AND (#iUNIT_NO = 1) THEN
       "DB440_MACHINE_ALARM_DECODING".ALARMS_UNIT_01.ST3_CLADDING.RHP_SEOC_ALARMS := FALSE;
       "DB440_MACHINE_ALARM_DECODING".ALARMS_UNIT_01.ST3_CLADDING.IS_SEOC_ALARMS := FALSE;
   END_IF;
   IF "DB2120_MPP_ITC_IPC".RESET_FAULTS AND (#iUNIT_NO = 2) THEN
       "DB440_MACHINE_ALARM_DECODING".ALARMS_UNIT_02.ST3_CLADDING.RHP_SEOC_ALARMS := FALSE;
       "DB440_MACHINE_ALARM_DECODING".ALARMS_UNIT_02.ST3_CLADDING.IS_SEOC_ALARMS := FALSE;
   END_IF;
END_REGION

REGION Network 32: LASER READY MODULE 1 IN TEST MODE ALARM
   RUNG wire#powerrail
      I_Contact( #iLASER_WARNING_LAP_ON )
      Contact( #iMACHINE_ON )
      Coil( #oALARM_LASER_MODULE_1_IN_TEST_MODE )
   END_RUNG
   // the same network as SCL:
   #oALARM_LASER_MODULE_1_IN_TEST_MODE := NOT #iLASER_WARNING_LAP_ON AND #iMACHINE_ON;
END_REGION

REGION Network 33: WARNING
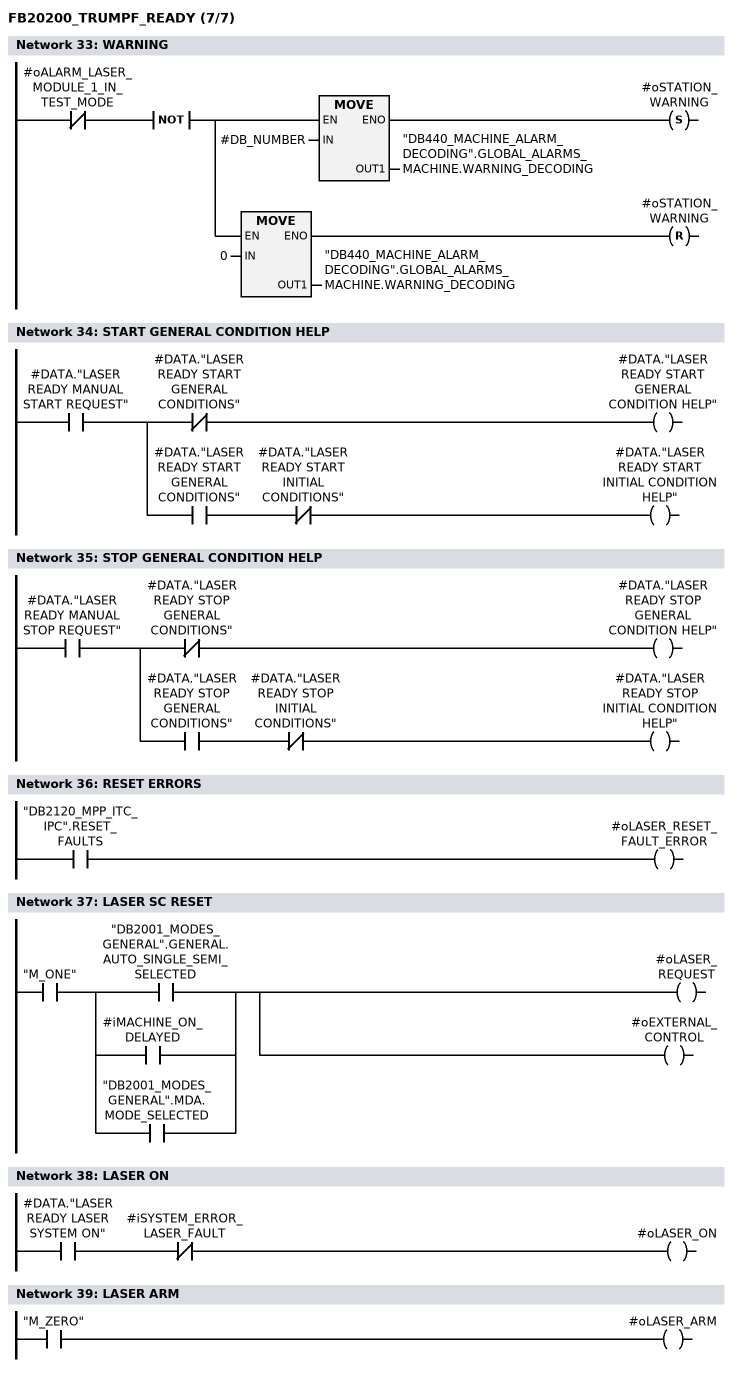
   RUNG wire#powerrail
      I_Contact( #oALARM_LASER_MODULE_1_IN_TEST_MODE )
      Not()
      wire#w1
      Move(in := #DB_NUMBER, out1 => "DB440_MACHINE_ALARM_DECODING".GLOBAL_ALARMS_MACHINE.WARNING_DECODING)
      S_Coil( #oSTATION_WARNING )
   END_RUNG
   RUNG wire#w1
      Move(in := 0, out1 => "DB440_MACHINE_ALARM_DECODING".GLOBAL_ALARMS_MACHINE.WARNING_DECODING)
      R_Coil( #oSTATION_WARNING )
   END_RUNG
   // the same network as SCL:
   IF NOT (NOT #oALARM_LASER_MODULE_1_IN_TEST_MODE) THEN
       "DB440_MACHINE_ALARM_DECODING".GLOBAL_ALARMS_MACHINE.WARNING_DECODING := #DB_NUMBER;
       #oSTATION_WARNING := TRUE;
       "DB440_MACHINE_ALARM_DECODING".GLOBAL_ALARMS_MACHINE.WARNING_DECODING := 0;
       #oSTATION_WARNING := FALSE;
   END_IF;
END_REGION

REGION Network 34: START GENERAL CONDITION HELP
   RUNG wire#powerrail
      Contact( #DATA."LASER READY MANUAL START REQUEST" )
      wire#w1
      I_Contact( #DATA."LASER READY START GENERAL CONDITIONS" )
      Coil( #DATA."LASER READY START GENERAL CONDITION HELP" )
   END_RUNG
   RUNG wire#w1
      Contact( #DATA."LASER READY START GENERAL CONDITIONS" )
      I_Contact( #DATA."LASER READY START INITIAL CONDITIONS" )
      Coil( #DATA."LASER READY START INITIAL CONDITION HELP" )
   END_RUNG
   // the same network as SCL:
   #DATA."LASER READY START GENERAL CONDITION HELP" := #DATA."LASER READY MANUAL START REQUEST" AND NOT #DATA."LASER READY START GENERAL CONDITIONS";
   #DATA."LASER READY START INITIAL CONDITION HELP" := #DATA."LASER READY MANUAL START REQUEST" AND #DATA."LASER READY START GENERAL CONDITIONS" AND NOT #DATA."LASER READY START INITIAL CONDITIONS";
END_REGION

REGION Network 35: STOP GENERAL CONDITION HELP
   RUNG wire#powerrail
      Contact( #DATA."LASER READY MANUAL STOP REQUEST" )
      wire#w1
      I_Contact( #DATA."LASER READY STOP GENERAL CONDITIONS" )
      Coil( #DATA."LASER READY STOP GENERAL CONDITION HELP" )
   END_RUNG
   RUNG wire#w1
      Contact( #DATA."LASER READY STOP GENERAL CONDITIONS" )
      I_Contact( #DATA."LASER READY STOP INITIAL CONDITIONS" )
      Coil( #DATA."LASER READY STOP INITIAL CONDITION HELP" )
   END_RUNG
   // the same network as SCL:
   #DATA."LASER READY STOP GENERAL CONDITION HELP" := #DATA."LASER READY MANUAL STOP REQUEST" AND NOT #DATA."LASER READY STOP GENERAL CONDITIONS";
   #DATA."LASER READY STOP INITIAL CONDITION HELP" := #DATA."LASER READY MANUAL STOP REQUEST" AND #DATA."LASER READY STOP GENERAL CONDITIONS" AND NOT #DATA."LASER READY STOP INITIAL CONDITIONS";
END_REGION

REGION Network 36: RESET ERRORS
   RUNG wire#powerrail
      Contact( "DB2120_MPP_ITC_IPC".RESET_FAULTS )
      Coil( #oLASER_RESET_FAULT_ERROR )
   END_RUNG
   // the same network as SCL:
   #oLASER_RESET_FAULT_ERROR := "DB2120_MPP_ITC_IPC".RESET_FAULTS;
END_REGION

REGION Network 37: LASER SC RESET
   RUNG wire#powerrail
      Contact( "M_ONE" )
      wire#w1
      Contact( "DB2001_MODES_GENERAL".GENERAL.AUTO_SINGLE_SEMI_SELECTED )
      wire#w2
      Coil( #oLASER_REQUEST )
   END_RUNG
   RUNG wire#w1
      Contact( #iMACHINE_ON_DELAYED )
   END_RUNG wire#w2
   RUNG wire#w1
      Contact( "DB2001_MODES_GENERAL".MDA.MODE_SELECTED )
   END_RUNG wire#w2
   RUNG wire#w2
      Coil( #oEXTERNAL_CONTROL )
   END_RUNG
   // the same network as SCL:
   #oLASER_REQUEST := "M_ONE" AND ("DB2001_MODES_GENERAL".GENERAL.AUTO_SINGLE_SEMI_SELECTED OR #iMACHINE_ON_DELAYED OR "DB2001_MODES_GENERAL".MDA.MODE_SELECTED);
   #oEXTERNAL_CONTROL := #oLASER_REQUEST;
END_REGION

REGION Network 38: LASER ON
   RUNG wire#powerrail
      Contact( #DATA."LASER READY LASER SYSTEM ON" )
      I_Contact( #iSYSTEM_ERROR_LASER_FAULT )
      Coil( #oLASER_ON )
   END_RUNG
   // the same network as SCL:
   #oLASER_ON := #DATA."LASER READY LASER SYSTEM ON" AND NOT #iSYSTEM_ERROR_LASER_FAULT;
END_REGION

REGION Network 39: LASER ARM
   RUNG wire#powerrail
      Contact( "M_ZERO" )
      Coil( #oLASER_ARM )
   END_RUNG
   // the same network as SCL:
   #oLASER_ARM := "M_ZERO";
END_REGION
END_FUNCTION_BLOCK
